	sInfraBool := Json.GetSymbolNameByAddress(
		nData := SIZEOF(GVL_TestSymbols.InfrastructureBool),
		pData := ADR(GVL_TestSymbols.InfrastructureBool),
		hrErrorCode => hr
	);
	sInfraLReal := Json.GetSymbolNameByAddress(
		nData := SIZEOF(GVL_TestSymbols.InfrastructureLReal),
		pData := ADR(GVL_TestSymbols.InfrastructureLReal),
		hrErrorCode => hr
	);
	sInput := Json.GetSymbolNameByAddress(
		nData := SIZEOF(GVL_TestSymbols.ModuleOne.InputBool),
		pData := ADR(GVL_TestSymbols.ModuleOne.InputBool),
		hrErrorCode => hr
	);
	sLongReal := Json.GetSymbolNameByAddress(
		nData := SIZEOF(GVL_TestSymbols.ModuleOne.LongRealValue),
		pData := ADR(GVL_TestSymbols.ModuleOne.LongRealValue),
		hrErrorCode => hr
	);
	AssertTrue(
		Condition := Manager.M_AddLink(
			SourceName := sInfraBool,
			TargetName := sInput,
			SourceDataType := E_ConfigDataType.Boolean,
			TargetDataType := E_ConfigDataType.Boolean,
			Phase := E_LinkPhase.InputToModule,
			HasTransform := FALSE,
			Scale := 1,
			Offset := 0
		),
		Message := 'Identical BOOL nodes must create a MEMCPY link.'
	);
	AssertTrue(
		Condition := Manager.M_AddLink(
			SourceName := sInfraLReal,
			TargetName := sLongReal,
			SourceDataType := E_ConfigDataType.Float64,
			TargetDataType := E_ConfigDataType.Float64,
			Phase := E_LinkPhase.InputToModule,
			HasTransform := TRUE,
			Scale := 2,
			Offset := 1
		),
		Message := 'Numeric transform link must be accepted.'
	);
	bInitialized := TRUE;
END_IF

// Act：Output phase 不得提前複製 Input link；Input phase 才套用兩種路徑。
GVL_TestSymbols.InfrastructureBool := TRUE;
GVL_TestSymbols.InfrastructureLReal := 10.0;
GVL_TestSymbols.ModuleOne.InputBool := FALSE;
GVL_TestSymbols.ModuleOne.LongRealValue := 0.0;
Manager.M_CyclicOutput();
AssertFalse(
	Condition := GVL_TestSymbols.ModuleOne.InputBool,
	Message := 'Wrong phase must not copy input data.'
);
Manager.M_CyclicInput();
AssertTrue(
	Condition := GVL_TestSymbols.ModuleOne.InputBool,
	Message := 'Input phase must copy BOOL data.'
);
AssertTrue(
	Condition := GVL_TestSymbols.ModuleOne.LongRealValue = 21.0,
	Message := 'Scale and offset must be applied in LREAL.'
);

TEST_FINISHED();
END_METHOD

METHOD ReadableNodeAndSingleWriterValidationAreExplicit
VAR_INST
	Manager : FB_LinkVariableManager;
	Json : FB_JsonReadWriteDataType;
	Config : ST_ModuleFileConfig;
	bInitialized : BOOL;
END_VAR
VAR
	sSource : STRING(255);
	sTarget : STRING(255);
	sModule : STRING(255);
	hr : HRESULT;
	nHandle : UINT;
	Raw : ST_ConfigRawValue;
	eRead : E_ConfigValueError;
	bOk : BOOL;
END_VAR
TEST('ReadableNodeAndSingleWriterValidationAreExplicit');

IF NOT bInitialized THEN
	Manager.M_BeginInfrastructureRegistration();
	Manager.M_RegisterInfrastructureNode(
		Variable := GVL_TestSymbols.InfrastructureBool,
		Access := E_VariableAccess.ReadOnly
	);
	Manager.M_SealInfrastructureRegistration();
	Manager.M_BeginModuleRegistration(
		Address := ADR(GVL_TestSymbols.ModuleTwo),
		Size := SIZEOF(GVL_TestSymbols.ModuleTwo),
		ModuleConfig := Config
	);
	Manager.M_RegisterModuleNode(
		Variable := GVL_TestSymbols.ModuleTwo.InputBool,
		Access := E_VariableAccess.ReadWrite
	);
	Manager.M_EndModuleRegistration(ModuleSymbol => sModule);
	sSource := Json.GetSymbolNameByAddress(
		nData := SIZEOF(GVL_TestSymbols.InfrastructureBool),
		pData := ADR(GVL_TestSymbols.InfrastructureBool),
		hrErrorCode => hr
	);
	sTarget := Json.GetSymbolNameByAddress(
		nData := SIZEOF(GVL_TestSymbols.ModuleTwo.InputBool),
		pData := ADR(GVL_TestSymbols.ModuleTwo.InputBool),
		hrErrorCode => hr
	);
	bInitialized := TRUE;
END_IF

AssertTrue(
	Condition := Manager.M_ResolveReadableNode(
		Name := sSource,
		ExpectedDataType := E_ConfigDataType.Boolean,
		NodeHandle => nHandle
	),
	Message := 'Readable registered source must resolve to a handle.'
);
GVL_TestSymbols.InfrastructureBool := TRUE;
AssertTrue(
	Condition := Manager.M_ReadNode(
		NodeHandle := nHandle,
		ExpectedDataType := E_ConfigDataType.Boolean,
		Value := Raw,
		ErrorCode => eRead
	),
	Message := 'Resolved handle must read its local value.'
);
AssertFalse(
	Condition := Manager.M_ReadNode(
		NodeHandle := 0,
		ExpectedDataType := E_ConfigDataType.Boolean,
		Value := Raw,
		ErrorCode => eRead
	),
	Message := 'Handle zero must be rejected.'
);
AssertTrue(
	Condition := eRead = E_ConfigValueError.InvalidNodeHandle,
	Message := 'Invalid handle must return a stable error code.'
);

AssertTrue(
	Condition := Manager.M_AddLink(
		SourceName := sSource,
		TargetName := sTarget,
		SourceDataType := E_ConfigDataType.Boolean,
		TargetDataType := E_ConfigDataType.Boolean,
		Phase := E_LinkPhase.InputToModule,
		HasTransform := FALSE,
		Scale := 1,
		Offset := 0
	),
	Message := 'First target writer must be accepted.'
);
AssertFalse(
	Condition := Manager.M_AddLink(
		SourceName := sSource,
		TargetName := sTarget,
		SourceDataType := E_ConfigDataType.Boolean,
		TargetDataType := E_ConfigDataType.Boolean,
		Phase := E_LinkPhase.ModuleToOutput,
		HasTransform := FALSE,
		Scale := 1,
		Offset := 0
	),
	Message := 'Second writer for the same target must be rejected.'
);

TEST_FINISHED();
END_METHOD

END_FUNCTION_BLOCK

// ---- POUs/Test Suites/Configuration/FB_ReferenceManagerTests.TcPOU
FUNCTION_BLOCK FB_ReferenceManagerTests EXTENDS TcUnit.FB_TestSuite

InvalidInterfacesAreRejectedBeforeRegistration();
RegisteredAdsSymbolCanBeResolved();

METHOD InvalidInterfacesAreRejectedBeforeRegistration
VAR_INST
	Manager : FB_ReferenceManager;
	NoProvider : FB_FakeBaseUnit;
	Missing : I_BaseUnit;
END_VAR
TEST('InvalidInterfacesAreRejectedBeforeRegistration');

// Assert：未綁定 interface 與未實作 I_AdsSymbolProvider 的 BaseUnit 都必須拒絕。
AssertFalse(
	Condition := Manager.M_RegisterReference(BaseUnit := Missing),
	Message := 'An unbound BaseUnit must be rejected.'
);
AssertFalse(
	Condition := Manager.M_RegisterReference(BaseUnit := NoProvider),
	Message := 'A BaseUnit without ADS metadata provider must be rejected.'
);

TEST_FINISHED();
END_METHOD

METHOD RegisteredAdsSymbolCanBeResolved
VAR_INST
	Manager : FB_ReferenceManager;
	Json : FB_JsonReadWriteDataType;
END_VAR
VAR
	Source : I_BaseUnit;
	Resolved : I_BaseUnit;
	sName : STRING(255);
	hr : HRESULT;
END_VAR
TEST('RegisteredAdsSymbolCanBeResolved');

// Arrange：使用具名 GVL instance，讓 runtime 可由 address/size 取得穩定 ADS symbol。
Source := GVL_TestSymbols.RegisteredBaseUnit;
sName := Json.GetSymbolNameByAddress(
	nData := SIZEOF(GVL_TestSymbols.RegisteredBaseUnit),
	pData := ADR(GVL_TestSymbols.RegisteredBaseUnit),
	hrErrorCode => hr
);
AssertTrue(
	Condition := (hr = 0) AND (sName <> ''),
	Message := 'Test BaseUnit must expose an ADS symbol.'
);

// Act / Assert。
AssertTrue(
	Condition := Manager.M_RegisterReference(BaseUnit := Source),
	Message := 'A symbol-backed BaseUnit must register.'
);
Resolved := Manager.M_Resolve(Name := sName);
AssertTrue(
	Condition := Resolved = Source,
	Message := 'Resolve must return the registered interface.'
);
Resolved := Manager.M_Resolve(Name := 'GVL_TestSymbols.DoesNotExist');
AssertTrue(
	Condition := (Resolved = 0) AND Manager.Error,
	Message := 'Unknown reference source must be explicit.'
);

TEST_FINISHED();
END_METHOD

END_FUNCTION_BLOCK

// ---- Fakes/FB_FakeBaseUnit.TcPOU
FUNCTION_BLOCK FB_FakeBaseUnit IMPLEMENTS I_BaseUnit

END_FUNCTION_BLOCK

// ---- POUs/Test Suites/Configuration/FB_ModuleReferenceBindingContextTests.TcPOU
FUNCTION_BLOCK FB_ModuleReferenceBindingContextTests EXTENDS TcUnit.FB_TestSuite

RequiredPortResolvesFromItsActualStorage();
OptionalMissingAndUnknownConfiguredKeysDiffer();
ScopeOrderingAndDuplicateTakePreserveFirstError();

METHOD RequiredPortResolvesFromItsActualStorage
VAR_INST
	Manager : FB_ReferenceManager;
	Context : FB_ModuleReferenceBindingContext;
	Json : FB_JsonReadWriteDataType;
	Config : ST_ModuleFileConfig;
END_VAR
VAR
	Source : I_BaseUnit;
	Resolved : I_BaseUnit;
	Bindings : I_ModuleReferenceBindings;
	sSource : STRING(255);
	sModule : STRING(255);
	sPort : STRING(80);
	sError : STRING(255);
	hr : HRESULT;
END_VAR
TEST('RequiredPortResolvesFromItsActualStorage');

// Arrange：註冊 BaseUnit source，並以實際 Module instance 的 ADS symbol 建立 scope。
Source := GVL_TestSymbols.RegisteredBaseUnit;
sSource := Json.GetSymbolNameByAddress(
	nData := SIZEOF(GVL_TestSymbols.RegisteredBaseUnit),
	pData := ADR(GVL_TestSymbols.RegisteredBaseUnit),
	hrErrorCode => hr
);
sModule := Json.GetSymbolNameByAddress(
	nData := SIZEOF(GVL_TestSymbols.ModuleOne),
	pData := ADR(GVL_TestSymbols.ModuleOne),
	hrErrorCode => hr
);
AssertTrue(
	Condition := Manager.M_RegisterReference(BaseUnit := Source),
	Message := 'Reference source must register.'
);
Config.ReferenceCount := 1;
Config.References[1].Name := 'BaseUnitPort';
Config.References[1].Source := sSource;
AssertTrue(
	Condition := Context.M_Begin(ModuleConfig := Config, ReferenceManager := Manager),
	Message := 'Binding session must begin.'
);
Bindings := Context;
AssertTrue(
	Condition := Bindings.M_SetModuleScope(ModuleSymbol := sModule, ErrorMessage => sError),
	Message := 'Module scope must be accepted once.'
);

// Act：即使 port 尚未綁定，ANY storage 仍可解析其相對名稱。
Resolved := Bindings.M_TakeRequired(
	Port := GVL_TestSymbols.ModuleOne.BaseUnitPort,
	PortName => sPort,
	ErrorMessage => sError
);
AssertTrue(
	Condition := (Resolved = Source) AND (sPort = 'BaseUnitPort'),
	Message := 'Required port must resolve by its actual storage name.'
);
AssertTrue(Condition := Context.M_End(), Message := 'All configured keys were consumed.');

TEST_FINISHED();
END_METHOD

METHOD OptionalMissingAndUnknownConfiguredKeysDiffer
VAR_INST
	OptionalContext : FB_ModuleReferenceBindingContext;
	UnknownContext : FB_ModuleReferenceBindingContext;
	Manager : FB_ReferenceManager;
	Json : FB_JsonReadWriteDataType;
	EmptyConfig : ST_ModuleFileConfig;
	UnknownConfig : ST_ModuleFileConfig;
END_VAR
VAR
	Bindings : I_ModuleReferenceBindings;
	Result : I_BaseUnit;
	sModule : STRING(255);
	sPort : STRING(80);
	sError : STRING(255);
	bPresent : BOOL;
	hr : HRESULT;
END_VAR
TEST('OptionalMissingAndUnknownConfiguredKeysDiffer');

sModule := Json.GetSymbolNameByAddress(
	nData := SIZEOF(GVL_TestSymbols.ModuleOne),
	pData := ADR(GVL_TestSymbols.ModuleOne),
	hrErrorCode => hr
);

// Optional omission 是合法結果：Present=FALSE、無錯誤，End 仍成功。
AssertTrue(
	Condition := OptionalContext.M_Begin(
		ModuleConfig := EmptyConfig,
		ReferenceManager := Manager
	),
	Message := 'Empty binding session must begin.'
);
Bindings := OptionalContext;
AssertTrue(
	Condition := Bindings.M_SetModuleScope(ModuleSymbol := sModule, ErrorMessage => sError),
	Message := 'Optional session needs a scope.'
);
Result := Bindings.M_TakeOptional(
	Port := GVL_TestSymbols.ModuleOne.BaseUnitPort,
	PortName => sPort,
	Present => bPresent,
	ErrorMessage => sError
);
AssertTrue(
	Condition := (Result = 0) AND NOT bPresent AND (sError = ''),
	Message := 'Missing optional key must be a clean omission.'
);
AssertTrue(
	Condition := OptionalContext.M_End(),
	Message := 'Optional omission must not leave an unknown key.'
);

// Configured key 若未被 adapter 消費，End 必須拒絕。
UnknownConfig.ReferenceCount := 1;
UnknownConfig.References[1].Name := 'UnknownPort';
UnknownConfig.References[1].Source := 'unused';
AssertTrue(
	Condition := UnknownContext.M_Begin(
		ModuleConfig := UnknownConfig,
		ReferenceManager := Manager
	),
	Message := 'Unknown-key session must begin.'
);
AssertFalse(
	Condition := UnknownContext.M_End(),
	Message := 'Unconsumed configured key must fail End.'
);
AssertTrue(
	Condition := UnknownContext.Error,
	Message := 'Unknown configured key must latch an error.'
);

TEST_FINISHED();
END_METHOD

METHOD ScopeOrderingAndDuplicateTakePreserveFirstError
VAR_INST
	Context : FB_ModuleReferenceBindingContext;
	Manager : FB_ReferenceManager;
	Config : ST_ModuleFileConfig;
	Json : FB_JsonReadWriteDataType;
END_VAR
VAR
	Bindings : I_ModuleReferenceBindings;
	Source : I_BaseUnit;
	Result : I_BaseUnit;
	sSource : STRING(255);
	sModule : STRING(255);
	sPort : STRING(80);
	sError : STRING(255);
	hr : HRESULT;
END_VAR
TEST('ScopeOrderingAndDuplicateTakePreserveFirstError');

Source := GVL_TestSymbols.RegisteredBaseUnit;
sSource := Json.GetSymbolNameByAddress(
	nData := SIZEOF(GVL_TestSymbols.RegisteredBaseUnit),
	pData := ADR(GVL_TestSymbols.RegisteredBaseUnit),
	hrErrorCode => hr
);
sModule := Json.GetSymbolNameByAddress(
	nData := SIZEOF(GVL_TestSymbols.ModuleOne),
	pData := ADR(GVL_TestSymbols.ModuleOne),
	hrErrorCode => hr
);
Manager.M_RegisterReference(BaseUnit := Source);
Config.ReferenceCount := 1;
Config.References[1].Name := 'BaseUnitPort';
Config.References[1].Source := sSource;
Context.M_Begin(ModuleConfig := Config, ReferenceManager := Manager);
Bindings := Context;
Bindings.M_SetModuleScope(ModuleSymbol := sModule, ErrorMessage => sError);
Result := Bindings.M_TakeRequired(
	Port := GVL_TestSymbols.ModuleOne.BaseUnitPort,
	PortName => sPort,
	ErrorMessage => sError
);
Result := Bindings.M_TakeRequired(
	Port := GVL_TestSymbols.ModuleOne.BaseUnitPort,
	PortName => sPort,
	ErrorMessage => sError
);
AssertTrue(
	Condition := Context.Error AND (FIND(Context.ErrorMessage, 'more than once') > 0),
	Message := 'Taking one configured key twice must fail explicitly.'
);

// 第一次錯誤鎖存後，後續 End 不可覆蓋診斷。
AssertFalse(
	Condition := Context.M_End(),
	Message := 'A failed binding session cannot end successfully.'
);
AssertTrue(
	Condition := FIND(Context.ErrorMessage, 'more than once') > 0,
	Message := 'The first binding error must be preserved.'
);

TEST_FINISHED();
END_METHOD

END_FUNCTION_BLOCK

// ---- POUs/Test Suites/Configuration/FB_ModuleTypeRegistryTests.TcPOU
FUNCTION_BLOCK FB_ModuleTypeRegistryTests EXTENDS TcUnit.FB_TestSuite

RegistrationResolveAndReplacementAreDeterministic();
CapacityAndClearFailuresAreExplicit();

METHOD CapacityAndClearFailuresAreExplicit
VAR_INST
	Registry : FB_ModuleTypeRegistry;
	Adapter : FB_FakeModuleConfigurationAdapter;
END_VAR
VAR
	nIndex : UINT;
	sName : T_ModuleTypeName;
	bOk : BOOL;
END_VAR
TEST('CapacityAndClearFailuresAreExplicit');

// Arrange：同一 adapter 可用不同 type name 填滿 registry。
FOR nIndex := 1 TO Param_Config.MaxModuleTypes DO
	sName := CONCAT('Type', UINT_TO_STRING(nIndex));
	bOk := Registry.M_Register(ModuleTypeName := sName, Adapter := Adapter);
END_FOR
AssertFalse(
	Condition := Registry.M_Register(ModuleTypeName := 'Overflow', Adapter := Adapter),
	Message := 'Registry entry beyond capacity must be rejected.'
);

// Act / Assert：adapter 的清除錯誤必須由 registry 原樣揭露。
Adapter.FailClear := TRUE;
AssertFalse(
	Condition := Registry.M_ClearAll(),
	Message := 'Adapter clear failure must fail ClearAll.'
);
AssertTrue(
	Condition := Registry.Error AND (Registry.ErrorMessage = 'Fake adapter clear failure.'),
	Message := 'ClearAll must preserve the adapter diagnostic.'
);

TEST_FINISHED();
END_METHOD

METHOD RegistrationResolveAndReplacementAreDeterministic
VAR_INST
	Registry : FB_ModuleTypeRegistry;
	AdapterOne : FB_FakeModuleConfigurationAdapter;
	AdapterTwo : FB_FakeModuleConfigurationAdapter;
	Resolved : I_ModuleConfigurationAdapter;
	pResolved : POINTER TO FB_FakeModuleConfigurationAdapter;
	EmptyAdapter : I_ModuleConfigurationAdapter;
END_VAR
VAR
	bResult : BOOL;
END_VAR
TEST('RegistrationResolveAndReplacementAreDeterministic');

// Arrange / Assert：名稱與 adapter 都是必要條件。
AssertFalse(
	Condition := Registry.M_Register(ModuleTypeName := '', Adapter := AdapterOne),
	Message := 'Empty module type name must be rejected.'
);
AssertFalse(
	Condition := Registry.M_Register(ModuleTypeName := 'Missing', Adapter := EmptyAdapter),
	Message := 'Unbound adapter must be rejected.'
);

// Act：同名第二次註冊應替換 adapter，不增加容量。
AssertTrue(
	Condition := Registry.M_Register(ModuleTypeName := 'TestModule', Adapter := AdapterOne),
	Message := 'A valid module type must register.'
);
Resolved := Registry.M_Resolve(ModuleTypeName := 'TestModule');
AssertTrue(
	Condition:= __QUERYPOINTER(Resolved, pResolved),
	Message:= 'Resolved adapter can not get pointer from interface.'
);
AssertTrue(
	Condition := pResolved = ADR(AdapterOne),
	Message := 'Resolve must return the registered adapter.'
);

AssertTrue(
	Condition := Registry.M_Register(ModuleTypeName := 'TestModule', Adapter := AdapterTwo),
	Message := 'Same-name registration must replace the adapter.'
);
Resolved := Registry.M_Resolve(ModuleTypeName := 'TestModule');
AssertTrue(
	Condition:= __QUERYPOINTER(Resolved, pResolved),
	Message:= 'Resolved adapter can not get pointer from interface.'
);
AssertTrue(
	Condition := pResolved = ADR(AdapterTwo),
	Message := 'Resolve must return the replacement adapter.'
);

Resolved := Registry.M_Resolve(ModuleTypeName := 'Unknown');
AssertTrue(
	Condition := (Resolved = 0) AND Registry.Error,
	Message := 'Unknown type must return an error and no adapter.'
);

TEST_FINISHED();
END_METHOD

END_FUNCTION_BLOCK

// ---- Fakes/FB_FakeModuleConfigurationAdapter.TcPOU
FUNCTION_BLOCK FB_FakeModuleConfigurationAdapter IMPLEMENTS I_ModuleConfigurationAdapter
VAR_INPUT
	FailClear : BOOL;
	FailPrepare : BOOL;
	FailApply : BOOL;
END_VAR
VAR_OUTPUT
	ClearCalls : UINT;
	PrepareCalls : UINT;
	ApplyCalls : UINT;
	LastSlot : UINT;
	LastRevision : UDINT;
END_VAR

METHOD PUBLIC M_ApplyRuntimeConfig : BOOL
VAR_INPUT
	Slot : UINT;
END_VAR
VAR_IN_OUT CONSTANT
	RuntimeConfig : ST_ModuleRuntimeConfig;
END_VAR
VAR_OUTPUT
	ErrorMessage : STRING(255);
END_VAR
ApplyCalls := ApplyCalls + 1;
LastSlot := Slot;
LastRevision := RuntimeConfig.Revision;
M_ApplyRuntimeConfig := NOT FailApply;
IF FailApply THEN
	ErrorMessage := 'Fake adapter apply failure.';
ELSE
	ErrorMessage := '';
END_IF
END_METHOD

METHOD PUBLIC M_ClearAllSlots : BOOL
VAR_OUTPUT
	ErrorMessage : STRING(255);
END_VAR
ClearCalls := ClearCalls + 1;
M_ClearAllSlots := NOT FailClear;
IF FailClear THEN
	ErrorMessage := 'Fake adapter clear failure.';
ELSE
	ErrorMessage := '';
END_IF
END_METHOD

METHOD PUBLIC M_IsSlotSupported : BOOL
VAR_INPUT
	Slot : UINT;
END_VAR
M_IsSlotSupported := (Slot >= 1) AND (Slot <= 2);
END_METHOD

METHOD PUBLIC M_PrepareInstance : BOOL
VAR_INPUT
	Slot : UINT;
	ReferenceBindings : I_ModuleReferenceBindings;
END_VAR
VAR_IN_OUT
	ModuleConfig : ST_ModuleFileConfig;
	LinkVariableManager : FB_LinkVariableManager;
END_VAR
VAR_OUTPUT
	ModuleSymbol : STRING(255);
	ErrorMessage : STRING(255);
END_VAR
VAR
	bOk : BOOL;
END_VAR
PrepareCalls := PrepareCalls + 1;
LastSlot := Slot;
ModuleSymbol := '';
ErrorMessage := '';
IF FailPrepare THEN
	ErrorMessage := 'Fake adapter prepare failure.';
	M_PrepareInstance := FALSE;
	RETURN;
END_IF
IF Slot = 1 THEN
	bOk := LinkVariableManager.M_BeginModuleRegistration(
		Address := ADR(GVL_TestSymbols.ModuleOne),
		Size := SIZEOF(GVL_TestSymbols.ModuleOne),
		ModuleConfig := ModuleConfig
	);
	bOk := LinkVariableManager.M_RegisterModuleNode(
		Variable := GVL_TestSymbols.ModuleOne.InputBool,
		Access := E_VariableAccess.ReadWrite
	);
	bOk := LinkVariableManager.M_RegisterModuleNode(
		Variable := GVL_TestSymbols.ModuleOne.OutputBool,
		Access := E_VariableAccess.ReadWrite
	);
	bOk := LinkVariableManager.M_RegisterModuleNode(
		Variable := GVL_TestSymbols.ModuleOne.LongRealValue,
		Access := E_VariableAccess.ReadWrite
	);
ELSE
	bOk := LinkVariableManager.M_BeginModuleRegistration(
		Address := ADR(GVL_TestSymbols.ModuleTwo),
		Size := SIZEOF(GVL_TestSymbols.ModuleTwo),
		ModuleConfig := ModuleConfig
	);
	bOk := LinkVariableManager.M_RegisterModuleNode(
		Variable := GVL_TestSymbols.ModuleTwo.InputBool,
		Access := E_VariableAccess.ReadWrite
	);
	bOk := LinkVariableManager.M_RegisterModuleNode(
		Variable := GVL_TestSymbols.ModuleTwo.OutputBool,
		Access := E_VariableAccess.ReadWrite
	);
	bOk := LinkVariableManager.M_RegisterModuleNode(
		Variable := GVL_TestSymbols.ModuleTwo.LongRealValue,
		Access := E_VariableAccess.ReadWrite
	);
END_IF
IF NOT bOk
	OR NOT LinkVariableManager.M_EndModuleRegistration(ModuleSymbol => ModuleSymbol) THEN
ErrorMessage := LinkVariableManager.ErrorMessage;
M_PrepareInstance := FALSE;
RETURN;
END_IF
M_PrepareInstance := TRUE;
END_METHOD

END_FUNCTION_BLOCK

// ---- POUs/Test Suites/Configuration/FB_ModuleConfigurationManagerTests.TcPOU
FUNCTION_BLOCK FB_ModuleConfigurationManagerTests EXTENDS TcUnit.FB_TestSuite

MissingConfigurationFileReturnsAStableError();
UnsupportedSchemaIsRejectedWhenRuntimeOptedIn();
LegacyAdsPortIsRejectedWhenRuntimeOptedIn();
DuplicateEnabledModuleIdIsRejectedWhenRuntimeOptedIn();
MalformedJsonIsRejectedWhenRuntimeOptedIn();
ValidFixtureAppliesOneRevisionWhenRuntimeOptedIn();

METHOD DuplicateEnabledModuleIdIsRejectedWhenRuntimeOptedIn
VAR_INST
	Manager : FB_ModuleConfigurationManager;
	Links : FB_LinkVariableManager;
	References : FB_ReferenceManager;
	Registry : FB_ModuleTypeRegistry;
	Adapter : FB_FakeModuleConfigurationAdapter;
	bPrepared : BOOL;
	nCycles : UINT;
END_VAR
VAR
	sPath : STRING(255);
END_VAR
IF NOT GVL_TestConfig.RunConfigurationFileRuntimeTests THEN
	RETURN;
END_IF
TEST('DuplicateEnabledModuleIdIsRejectedWhenRuntimeOptedIn');

IF NOT bPrepared THEN
	// Arrange：先滿足 infrastructure 與 adapter 前置條件，讓驗證能走到 ModuleId 唯一性規則。
	Links.M_BeginInfrastructureRegistration();
	Links.M_SealInfrastructureRegistration();
	Registry.M_Register(ModuleTypeName := 'TestModule', Adapter := Adapter);
	bPrepared := TRUE;
END_IF
sPath := CONCAT(GVL_TestConfig.ConfigurationFixtureRoot, 'duplicate-enabled-id.json');
// Act
Manager(
	Execute := TRUE,
	FilePath := sPath,
	LinkVariableManager := Links,
	ReferenceManager := References,
	ModuleTypeRegistry := Registry
);
nCycles := nCycles + 1;
IF Manager.Error THEN
	// Assert
	AssertTrue(
		Condition := Manager.ErrorMessage = 'Duplicate enabled module ID in configuration.',
		Message := 'Enabled ModuleId must be globally unique.'
	);
	AssertTrue(
		Condition := Adapter.ApplyCalls = 0,
		Message := 'Duplicate ModuleId must fail before adapter apply.'
	);
	nCycles := 0;
	TEST_FINISHED();
ELSIF nCycles > 1000 THEN
	AssertTrue(
		Condition := FALSE,
		Message := 'Duplicate-ID fixture timed out; verify fixture deployment.'
	);
	nCycles := 0;
	TEST_FINISHED();
END_IF
END_METHOD

METHOD LegacyAdsPortIsRejectedWhenRuntimeOptedIn
VAR_INST
	Manager : FB_ModuleConfigurationManager;
	Links : FB_LinkVariableManager;
	References : FB_ReferenceManager;
	Registry : FB_ModuleTypeRegistry;
	nCycles : UINT;
END_VAR
VAR
	sPath : STRING(255);
END_VAR
IF NOT GVL_TestConfig.RunConfigurationFileRuntimeTests THEN
	RETURN;
END_IF
TEST('LegacyAdsPortIsRejectedWhenRuntimeOptedIn');

// Arrange：schemaVersion 4 明確禁止舊版 adsPort 欄位。
sPath := CONCAT(GVL_TestConfig.ConfigurationFixtureRoot, 'legacy-ads-port.json');
// Act
Manager(
	Execute := TRUE,
	FilePath := sPath,
	LinkVariableManager := Links,
	ReferenceManager := References,
	ModuleTypeRegistry := Registry
);
nCycles := nCycles + 1;
IF Manager.Error THEN
	// Assert
	AssertTrue(
		Condition :=
			Manager.ErrorMessage =
			'adsPort is not supported by schemaVersion 4; configured values use registered local nodes.',
		Message := 'Legacy adsPort must be rejected with the documented diagnostic.'
	);
	nCycles := 0;
	TEST_FINISHED();
ELSIF nCycles > 1000 THEN
	AssertTrue(
		Condition := FALSE,
		Message := 'Legacy-adsPort fixture timed out; verify fixture deployment.'
	);
	nCycles := 0;
	TEST_FINISHED();
END_IF
END_METHOD

METHOD MalformedJsonIsRejectedWhenRuntimeOptedIn
VAR_INST
	Manager : FB_ModuleConfigurationManager;
	Links : FB_LinkVariableManager;
	References : FB_ReferenceManager;
	Registry : FB_ModuleTypeRegistry;
	nCycles : UINT;
END_VAR
VAR
	sPath : STRING(255);
END_VAR
IF NOT GVL_TestConfig.RunConfigurationFileRuntimeTests THEN
	RETURN;
END_IF
TEST('MalformedJsonIsRejectedWhenRuntimeOptedIn');

// Arrange：fixture 故意缺少合法的陣列結尾；副檔名保留 .invalid，避免被 JSON lint 誤當有效資料。
sPath := CONCAT(GVL_TestConfig.ConfigurationFixtureRoot, 'malformed.json.invalid');
// Act
Manager(
	Execute := TRUE,
	FilePath := sPath,
	LinkVariableManager := Links,
	ReferenceManager := References,
	ModuleTypeRegistry := Registry
);
nCycles := nCycles + 1;
IF Manager.Error THEN
	
	// 下一個 scan 才會關閉 Busy 的訊號
	Manager(
		Execute := TRUE,
		FilePath := sPath,
		LinkVariableManager := Links,
		ReferenceManager := References,
		ModuleTypeRegistry := Registry
	);
	
	// Assert：parser HRESULT 可能因 runtime 版本不同；穩定契約是 Error、非 Ready、且有診斷內容。
	AssertFalse(
		Condition := Manager.Ready OR Manager.Busy,
		Message := 'Malformed JSON must end in Error only.'
	);
	AssertTrue(
		Condition := Manager.ErrorMessage <> '',
		Message := 'Malformed JSON must expose a diagnostic message.'
	);
	nCycles := 0;
	TEST_FINISHED();
ELSIF nCycles > 1000 THEN
	AssertTrue(
		Condition := FALSE,
		Message := 'Malformed-JSON fixture timed out; verify fixture deployment.'
	);
	nCycles := 0;
	TEST_FINISHED();
END_IF
END_METHOD

METHOD MissingConfigurationFileReturnsAStableError
VAR_INST
	Manager : FB_ModuleConfigurationManager;
	Links : FB_LinkVariableManager;
	References : FB_ReferenceManager;
	Registry : FB_ModuleTypeRegistry;
	nCycles : UINT;
END_VAR
TEST('MissingConfigurationFileReturnsAStableError');

// Arrange / Act：以必定不存在的 fixture 路徑維持 Execute，高階 JSON loader 可能需要多個 PLC scan 才完成。
Manager(
	Execute := TRUE,
	FilePath := 'C:\ProgramData\RobustSolution\Tests\does-not-exist.json',
	LinkVariableManager := Links,
	ReferenceManager := References,
	ModuleTypeRegistry := Registry
);
nCycles := nCycles + 1;

IF Manager.Error THEN
	// 實作當 Error 發生時，下一個 scan 才會將 Busy 設為 False
	Manager(
		Execute := TRUE,
		FilePath := 'C:\ProgramData\RobustSolution\Tests\does-not-exist.json',
		LinkVariableManager := Links,
		ReferenceManager := References,
		ModuleTypeRegistry := Registry
	);

	// Assert：I/O error 必須結束 Busy 並提供固定診斷。
	AssertFalse(
		Condition := Manager.Busy OR Manager.Ready,
		Message := 'A missing file must end in Error only.'
	);
	AssertTrue(
		Condition := Manager.ErrorMessage =
			'Unable to load the UTF-8 JSON module configuration file.',
		Message := 'Missing file must expose the documented diagnostic.'
	);
	nCycles := 0;
	TEST_FINISHED();
ELSIF nCycles > 1000 THEN
	AssertTrue(
		Condition := FALSE,
		Message := 'Configuration file error did not complete within 1000 scans.'
	);
	nCycles := 0;
	TEST_FINISHED();
END_IF
END_METHOD

METHOD UnsupportedSchemaIsRejectedWhenRuntimeOptedIn
VAR_INST
	Manager : FB_ModuleConfigurationManager;
	Links : FB_LinkVariableManager;
	References : FB_ReferenceManager;
	Registry : FB_ModuleTypeRegistry;
	nCycles : UINT;
END_VAR
VAR
	sPath : STRING(255);
END_VAR
IF NOT GVL_TestConfig.RunConfigurationFileRuntimeTests THEN
	RETURN;
END_IF
TEST('UnsupportedSchemaIsRejectedWhenRuntimeOptedIn');

// Arrange：fixture 使用 framework 不支援的 schemaVersion 3。
sPath := CONCAT(GVL_TestConfig.ConfigurationFixtureRoot, 'unsupported-schema.json');
// Act：檔案解析是非同步流程，因此跨 scan 保持 Execute。
Manager(
	Execute := TRUE,
	FilePath := sPath,
	LinkVariableManager := Links,
	ReferenceManager := References,
	ModuleTypeRegistry := Registry
);
nCycles := nCycles + 1;
IF Manager.Error THEN
	// Assert：錯誤必須停在 schema 驗證，不可進入套用階段。
	AssertTrue(
		Condition := Manager.ErrorMessage = 'Unsupported module configuration schemaVersion.',
		Message := 'Unsupported schema must return its documented diagnostic.'
	);
	nCycles := 0;
	TEST_FINISHED();
ELSIF nCycles > 1000 THEN
	AssertTrue(
		Condition := FALSE,
		Message := 'Unsupported-schema fixture timed out; verify fixture deployment.'
	);
	nCycles := 0;
	TEST_FINISHED();
END_IF
END_METHOD

METHOD ValidFixtureAppliesOneRevisionWhenRuntimeOptedIn
VAR_INST
	Manager : FB_ModuleConfigurationManager;
	Links : FB_LinkVariableManager;
	References : FB_ReferenceManager;
	Registry : FB_ModuleTypeRegistry;
	Adapter : FB_FakeModuleConfigurationAdapter;
	bPrepared : BOOL;
	nCycles : UINT;
END_VAR
VAR
	sPath : STRING(255);
END_VAR
// RuntimeDependent：fixture 未部署時不註冊此 case，避免將環境缺失算成產品失敗。
IF NOT GVL_TestConfig.RunConfigurationFileRuntimeTests THEN
	RETURN;
END_IF
TEST('ValidFixtureAppliesOneRevisionWhenRuntimeOptedIn');

IF NOT bPrepared THEN
	// Arrange：Configuration Manager 要求 infrastructure 已 seal，並有可解析的 Module adapter。
	Links.M_BeginInfrastructureRegistration();
	Links.M_SealInfrastructureRegistration();
	Registry.M_Register(ModuleTypeName := 'TestModule', Adapter := Adapter);
	bPrepared := TRUE;
END_IF
sPath := CONCAT(GVL_TestConfig.ConfigurationFixtureRoot, 'valid-minimal.json');
Manager(
	Execute := TRUE,
	FilePath := sPath,
	LinkVariableManager := Links,
	ReferenceManager := References,
	ModuleTypeRegistry := Registry
);
nCycles := nCycles + 1;

IF Manager.Ready THEN
	
	// 下一個 scan 才會關閉 Busy 的訊號
	Manager(
		Execute := TRUE,
		FilePath := sPath,
		LinkVariableManager := Links,
		ReferenceManager := References,
		ModuleTypeRegistry := Registry
	);

	AssertFalse(
		Condition := Manager.Error OR Manager.Busy,
		Message := 'Valid fixture must finish Ready.'
	);
	AssertTrue(
		Condition :=
			(Adapter.PrepareCalls = 1)
			AND (Adapter.ApplyCalls = 1)
			AND (Adapter.LastSlot = 1)
			AND (Adapter.LastRevision = 1),
		Message := 'Valid fixture must prepare and apply exactly one runtime revision.'
	);
	nCycles := 0;
	TEST_FINISHED();
ELSIF Manager.Error OR (nCycles > 1000) THEN
	AssertTrue(
		Condition := FALSE,
		Message :=
			'Valid runtime fixture failed or timed out; verify deployment and installed Framework library.'
	);
	nCycles := 0;
	TEST_FINISHED();
END_IF
END_METHOD

END_FUNCTION_BLOCK

// ---- POUs/Test Suites/Configuration/FB_ApplicationConfigRootTests.TcPOU
FUNCTION_BLOCK FB_ApplicationConfigRootTests EXTENDS TcUnit.FB_TestSuite
VAR
	_ConfigRoot : FB_TestApplicationConfigRoot;
END_VAR

RegistrationHooksRunOnceInOrderAndLatchFailure();
ReadyCycleCopiesInputRunsModuleAndCopiesOutput();

METHOD RegistrationHooksRunOnceInOrderAndLatchFailure
TEST('RegistrationHooksRunOnceInOrderAndLatchFailure');

_ConfigRoot.Run();

AssertTrue(
	Condition := (_ConfigRoot.IoRegistrationCalls = 1)
		AND (_ConfigRoot.BaseUnitRegistrationCalls = 1)
		AND (_ConfigRoot.ModuleTypeRegistrationCalls = 1),
	Message := 'The three application registration hooks must each run once.');
AssertTrue(
	Condition := _ConfigRoot.RegistrationOrderValid,
	Message := 'Registration hooks must run in IO, BaseUnit, Module Type order.');
AssertTrue(
	Condition := _ConfigRoot.Error
		AND NOT _ConfigRoot.Ready
		AND (_ConfigRoot.ErrorCode = 0)
		AND (_ConfigRoot.ErrorMessage = 'A Module Type name and adapter are required.'),
	Message :=
		'The first registration failure must be exposed by the ConfigRoot properties.');

// A second cycle must neither retry registration nor enter configuration loading.
_ConfigRoot.Run();
AssertTrue(
	Condition := (_ConfigRoot.IoRegistrationCalls = 1)
		AND (_ConfigRoot.BaseUnitRegistrationCalls = 1)
		AND (_ConfigRoot.ModuleTypeRegistrationCalls = 1),
	Message := 'A latched startup failure must not retry application registration.');

// The public Run seam is gated by Ready.
AssertTrue(
	Condition := _ConfigRoot.ModuleCycleCalls = 0,
	Message :=
		'Module polling must remain disabled after configuration initialization fails.');

TEST_FINISHED();
END_METHOD

METHOD ReadyCycleCopiesInputRunsModuleAndCopiesOutput
VAR_INST
	Root : FB_TestApplicationConfigRoot;
	nCycles : UINT;
END_VAR
// RuntimeDependent：需將 library parameter 的 ModuleConfigFilePath 指向 application-root.json。
IF NOT GVL_TestConfig.RunConfigurationFileRuntimeTests THEN
	RETURN;
END_IF
TEST('ReadyCycleCopiesInputRunsModuleAndCopiesOutput');

// Arrange：使用有效 adapter，並準備可辨識的 input/output 初值。
Root.UseValidModuleTypeRegistration := TRUE;
GVL_TestSymbols.InfrastructureBool := TRUE;
GVL_TestSymbols.InfrastructureOutputBool := FALSE;

// Act：Config loader 可能跨多個 scan；Ready 後同一個 Run 會依 input、Module、output 的順序執行。
Root.Run();
nCycles := nCycles + 1;
IF Root.Ready THEN
	// Assert：hook 看到 input-copy 結果，外部節點看到 hook 產生的 output-copy 結果。
	AssertTrue(
		Condition := Root.ModuleObservedInput,
		Message := 'Input mapping must complete before the Module hook runs.'
	);
	AssertTrue(
		Condition := GVL_TestSymbols.InfrastructureOutputBool,
		Message := 'Output mapping must run after the Module hook.'
	);
	AssertTrue(
		Condition := (Root.ModuleCycleCalls > 0) AND (LEN(Root.LastSystemUtcDateTime) = 17),
		Message := 'Ready cycle must run Modules with an updated UTC context.'
	);
	AssertTrue(
		Condition := Root.LastHeartbeatTimeout = Param_Config.ModuleHeartbeat_Timeout,
		Message := 'SystemContext must carry the configured heartbeat timeout.'
	);
	nCycles := 0;
	TEST_FINISHED();
ELSIF Root.Error OR (nCycles > 1000) THEN
	AssertTrue(
		Condition := FALSE,
		Message :=
			'Application root fixture failed or timed out; verify library parameter and fixture deployment.'
	);
	nCycles := 0;
	TEST_FINISHED();
END_IF
END_METHOD

END_FUNCTION_BLOCK

// ---- Fakes/FB_TestApplicationConfigRoot.TcPOU
FUNCTION_BLOCK FB_TestApplicationConfigRoot EXTENDS FB_ApplicationConfigRoot
VAR_INPUT
	UseValidModuleTypeRegistration : BOOL;
END_VAR
VAR_OUTPUT
	IoRegistrationCalls : UINT;
	BaseUnitRegistrationCalls : UINT;
	ModuleTypeRegistrationCalls : UINT;
	ModuleCycleCalls : UINT;
	RegistrationOrderValid : BOOL := TRUE;
	ModuleObservedInput : BOOL;
	LastSystemUtcDateTime : STRING(20);
	LastHeartbeatTimeout : TIME;
END_VAR
VAR
	_nRegistrationStep : UINT;
	_Adapter : FB_FakeModuleConfigurationAdapter;
END_VAR

METHOD PROTECTED H_RegisterBaseUnits
BaseUnitRegistrationCalls := BaseUnitRegistrationCalls + 1;
_nRegistrationStep := _nRegistrationStep + 1;
RegistrationOrderValid := RegistrationOrderValid AND (_nRegistrationStep = 2);
M_RegisterBaseUnit(BaseUnit := GVL_TestSymbols.RegisteredBaseUnit);
END_METHOD

METHOD PROTECTED H_RegisterIo
IoRegistrationCalls := IoRegistrationCalls + 1;
_nRegistrationStep := _nRegistrationStep + 1;
RegistrationOrderValid := RegistrationOrderValid AND (_nRegistrationStep = 1);
M_RegisterIoNode(
	Variable := GVL_TestSymbols.InfrastructureBool,
	Access := E_VariableAccess.ReadOnly);
M_RegisterIoNode(
	Variable := GVL_TestSymbols.InfrastructureOutputBool,
	Access := E_VariableAccess.WriteOnly);
END_METHOD

METHOD PROTECTED H_RegisterModuleTypes
ModuleTypeRegistrationCalls := ModuleTypeRegistrationCalls + 1;
_nRegistrationStep := _nRegistrationStep + 1;
RegistrationOrderValid := RegistrationOrderValid AND (_nRegistrationStep = 3);

IF UseValidModuleTypeRegistration THEN
	// Runtime-dependent success seam: the fixture resolves this adapter by name.
	M_RegisterModuleType(ModuleTypeName := 'TestModule', Adapter := _Adapter);
ELSE
	// Deterministic failure seam: do not touch a target-dependent JSON file.
	M_RegisterModuleType(ModuleTypeName := '', Adapter := 0);
END_IF
END_METHOD

METHOD PROTECTED H_RunModules
VAR_INPUT
	VariableNodeReader : I_VariableNodeReader;
END_VAR
VAR_IN_OUT CONSTANT
	SystemContext : ST_SystemContext;
END_VAR
ModuleCycleCalls := ModuleCycleCalls + 1;
// 記錄 input-copy 已在 Module hook 前完成，並產生一筆 output-copy 可觀察值。
ModuleObservedInput := GVL_TestSymbols.ModuleOne.InputBool;
GVL_TestSymbols.ModuleOne.OutputBool := TRUE;
LastSystemUtcDateTime := SystemContext.UtcDateTime;
LastHeartbeatTimeout := SystemContext.ModuleHeartbeatTimeout;
END_METHOD

END_FUNCTION_BLOCK

// ---- Fakes/FB_FakeModuleReferenceBindings.TcPOU
FUNCTION_BLOCK FB_FakeModuleReferenceBindings IMPLEMENTS I_ModuleReferenceBindings
VAR_OUTPUT
	ModuleScope : STRING(255);
	ScopeSetCount : UINT;
	TakeCount : UINT;
	TakenAddresses : ARRAY[1..2] OF PVOID;
	TakenSizes : ARRAY[1..2] OF DINT;
END_VAR
VAR
	_RequiredResults : ARRAY[1..2] OF I_BaseUnit;
END_VAR

METHOD PUBLIC M_SetRequiredResult
VAR_INPUT
	BaseUnit : I_BaseUnit;
END_VAR
_RequiredResults[1] := BaseUnit;
_RequiredResults[2] := BaseUnit;
END_METHOD

METHOD PUBLIC M_TakeOptional : I_BaseUnit
VAR_INPUT
	Port : ANY;
END_VAR
VAR_OUTPUT
	PortName : STRING(80);
	Present : BOOL;
	ErrorMessage : STRING(255);
END_VAR
TakeCount := TakeCount + 1;
PortName := 'FakePort';
ErrorMessage := '';
IF TakeCount <= 2 THEN
	TakenAddresses[TakeCount] := Port.pValue;
	TakenSizes[TakeCount] := Port.diSize;
END_IF
M_TakeOptional := 0;
Present := FALSE;
END_METHOD

METHOD PUBLIC M_TakeRequired : I_BaseUnit
VAR_INPUT
	Port : ANY;
END_VAR
VAR_OUTPUT
	PortName : STRING(80);
	ErrorMessage : STRING(255);
END_VAR
TakeCount := TakeCount + 1;
PortName := 'FakePort';
ErrorMessage := '';
IF TakeCount <= 2 THEN
	TakenAddresses[TakeCount] := Port.pValue;
	TakenSizes[TakeCount] := Port.diSize;
END_IF
M_TakeRequired := 0;
IF TakeCount <= 2 THEN
	M_TakeRequired := _RequiredResults[TakeCount];
END_IF
IF M_TakeRequired = 0 THEN
	ErrorMessage := 'Injected required reference failure.';
END_IF
END_METHOD

METHOD PUBLIC M_SetRequiredResults
VAR_INPUT
	First : I_BaseUnit;
	Second : I_BaseUnit;
END_VAR
_RequiredResults[1] := First;
_RequiredResults[2] := Second;
END_METHOD

METHOD PUBLIC M_SetModuleScope : BOOL
VAR_INPUT
	ModuleSymbol : STRING(255);
END_VAR
VAR_OUTPUT
	ErrorMessage : STRING(255);
END_VAR
ModuleScope := ModuleSymbol;
ScopeSetCount := ScopeSetCount + 1;
TakeCount := 0;
MEMSET(ADR(TakenAddresses), 0, SIZEOF(TakenAddresses));
MEMSET(ADR(TakenSizes), 0, SIZEOF(TakenSizes));
ErrorMessage := '';
M_SetModuleScope := ModuleSymbol <> '';
END_METHOD

END_FUNCTION_BLOCK

// ---- Fakes/FB_ReferencePortFixture.TcPOU
FUNCTION_BLOCK FB_ReferencePortFixture
VAR_INPUT
	AxisOne : I_Axis_BaseUnit;
	AxisTwo : I_Axis_BaseUnit;
	OptionalAxis : I_Axis_BaseUnit;
	Nested : ST_ReferencePortTestBranch;
	BranchWithAnIntentionallyLongNameForReferenceTests : ST_ReferencePortTestBranch;
END_VAR

END_FUNCTION_BLOCK
